{attribute 'qualified_only'}
{attribute 'to_string'}
{attribute 'strict'}
TYPE E_DATA_CTRL :
(
  NULL,
	INIT  := 10,
  READ  := 20,
  WRITE := 30
)UINT;
END_TYPE

(* stored: Version 1.1.0.1, ProductVersion 3.1.4026.18
   DUT E_DATA_CTRL: Id {952fab49-9c02-4003-b3b1-ae8430162ba4} *)
